(*
Standard way to control assests in system
*)
FUNCTION_BLOCK ABSTRACT FB_PackMLControl
VAR_INPUT
END_VAR
VAR_OUTPUT
END_VAR
VAR
	state_idle : DINT;
	state_starting : DINT;
	state_execute : DINT;	
	start : BOOL;
	complete : BOOL;
	stateMachineResult : HResult;
END_VAR

METHOD PUBLIC ABSTRACT M_Aborted : HResult
VAR_INPUT
END_VAR
END_METHOD

METHOD PUBLIC ABSTRACT M_Aborting : HResult
VAR_INPUT
END_VAR
END_METHOD

METHOD PUBLIC ABSTRACT M_Complete : HResult
VAR_INPUT
END_VAR
VAR_OUTPUT
	abort : BOOL;
END_VAR
END_METHOD

METHOD PUBLIC ABSTRACT M_Completing : HREsult
VAR_INPUT
END_VAR
VAR_OUTPUT
	abort : BOOL;	
	stop : BOOL;
END_VAR
END_METHOD

METHOD PUBLIC ABSTRACT M_Execute : HResult
VAR_INPUT
	lastResult : HResult;
END_VAR
VAR_OUTPUT
	stop : BOOL;
	suspend : BOOL;
	hold : BOOL;
END_VAR
END_METHOD

METHOD PUBLIC ABSTRACT M_Held : HResult
VAR_INPUT
END_VAR
VAR_OUTPUT
	abort : BOOL;
	stop : BOOL;
END_VAR
END_METHOD

METHOD PUBLIC ABSTRACT M_Holding : HResult
VAR_INPUT
END_VAR
VAR_OUTPUT
	abort : BOOL;
	stop : BOOL;
END_VAR
END_METHOD

METHOD PUBLIC ABSTRACT M_Idle : HResult
VAR_INPUT
	lastResult : HResult;
END_VAR
VAR_OUTPUT
	abort : BOOL;
END_VAR
END_METHOD

METHOD PUBLIC ABSTRACT M_Resetting : HResult
VAR_INPUT
END_VAR
VAR_OUTPUT
	abort : BOOL;
	stop : BOOL;
END_VAR
END_METHOD

METHOD ABSTRACT M_Starting : HResult
VAR_INPUT
	lastResult : HResult;
END_VAR
VAR_OUTPUT
	abort : BOOL;
	stop : BOOL;
END_VAR
END_METHOD

METHOD PUBLIC ABSTRACT M_Stopped : HResult
VAR_INPUT
END_VAR
VAR_OUTPUT
	abort : BOOL;
END_VAR
END_METHOD

METHOD PUBLIC ABSTRACT M_Stopping : HResult
VAR_INPUT
END_VAR
VAR_OUTPUT
	abort : BOOL;
END_VAR
END_METHOD

METHOD PUBLIC ABSTRACT M_Suspended : HREsult
VAR_INPUT
END_VAR
VAR_OUTPUT
	abort : BOOL;
	stop : BOOL;
END_VAR
END_METHOD

METHOD PUBLIC ABSTRACT M_Suspending : HREsult
VAR_INPUT
END_VAR
VAR_OUTPUT
	abort : BOOL;
	stop : BOOL;
END_VAR
END_METHOD

METHOD PUBLIC ABSTRACT M_Un_Holding : HREsult
VAR_INPUT
END_VAR
VAR_OUTPUT
	abort : BOOL;
	stop : BOOL;
END_VAR
END_METHOD

METHOD PUBLIC ABSTRACT M_Un_Suspending : HREsult
VAR_INPUT
END_VAR
VAR_OUTPUT
	abort : BOOL;
	stop : BOOL;
END_VAR
END_METHOD

END_FUNCTION_BLOCK

(* stored: Version 1.1.0.1, ProductVersion 3.1.4024.12
   POU FB_PackMLControl: Id {61f7caa2-4ae2-4c52-ad20-bbdcfbe3e126}, SpecialFunc None
   Method M_Aborted: Id {953651d1-1c27-47e8-b880-20f5ea5520b9}
   Method M_Aborting: Id {1d5eb2f7-6d29-4d55-a7fc-67485706fbfc}
   Method M_Complete: Id {144f328d-5a96-4fd8-b49f-8b1cb5677afc}
   Method M_Completing: Id {aa4afca2-d4dc-438c-b0db-f8757335e3e8}
   Method M_Execute: Id {6d6c0d6f-162d-4964-b62c-51432b81664e}
   Method M_Held: Id {c018b924-2b76-445b-b007-e5482a3f1ede}
   Method M_Holding: Id {c9d2e81a-8ff8-45f4-9629-4792d830da49}
   Method M_Idle: Id {35d02f5b-8116-4985-857c-a6782823d22b}
   Method M_Resetting: Id {25f473c0-0dc0-4b69-aa09-6d6e0035ab3f}
   Method M_Starting: Id {f2f0aab8-8019-40af-ab0e-d4f9bae5be2d}
   Method M_Stopped: Id {a7431208-e9de-4c9c-87c1-3d3873fb997a}
   Method M_Stopping: Id {114ac1ae-6d83-4f7b-a35b-600ac2a46a2a}
   Method M_Suspended: Id {7927b8cf-8b2b-48ce-a526-32e3ccc9d11e}
   Method M_Suspending: Id {98d41089-f404-4bff-9508-f47765def391}
   Method M_Un_Holding: Id {ab65c218-0d63-44f3-9ba1-214a21d6d1c7}
   Method M_Un_Suspending: Id {22328fe1-193a-490d-9291-313194c1fa12} *)
